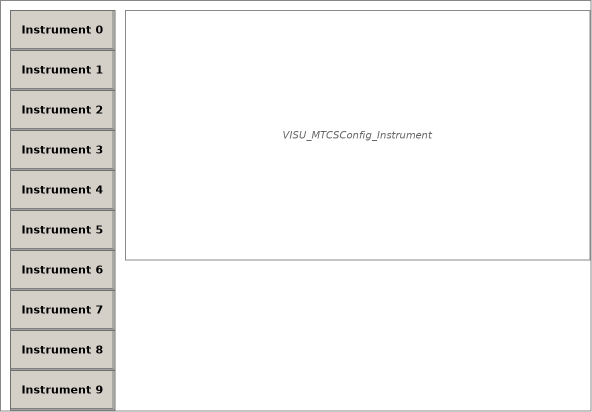
VISUALIZATION VISU_MTCSConfig_Instruments  // 592x412
VAR_IN_OUT
    active : MTCSInstrumentsConfig;
    editable : MTCSInstrumentsConfig;
	currentPosition : INT;
END_VAR
    Button (10,10 105x40), "Instrument 0", pressed state: currentPosition = 0
        OnMouseClick: execute { currentPosition := 0; }
    Button (10,50 105x40), "Instrument 1", pressed state: currentPosition = 1
        OnMouseClick: execute { currentPosition := 1; }
    Button (10,90 105x40), "Instrument 2", pressed state: currentPosition = 2
        OnMouseClick: execute { currentPosition := 2; }
    Button (10,130 105x40), "Instrument 3", pressed state: currentPosition = 3
        OnMouseClick: execute { currentPosition := 3; }
    Button (10,170 105x40), "Instrument 4", pressed state: currentPosition = 4
        OnMouseClick: execute { currentPosition := 4; }
    Button (10,210 105x40), "Instrument 5", pressed state: currentPosition = 5
        OnMouseClick: execute { currentPosition := 5; }
    Button (10,250 105x40), "Instrument 6", pressed state: currentPosition = 6
        OnMouseClick: execute { currentPosition := 6; }
    Button (10,290 105x40), "Instrument 7", pressed state: currentPosition = 7
        OnMouseClick: execute { currentPosition := 7; }
    Button (10,330 105x40), "Instrument 8", pressed state: currentPosition = 8
        OnMouseClick: execute { currentPosition := 8; }
    Button (10,370 105x40), "Instrument 9", pressed state: currentPosition = 9
        OnMouseClick: execute { currentPosition := 9; }
    Frame (125,10 465x250), frame switch variable: currentPosition
        shows VISU_MTCSConfig_Instrument(active := active.instrument0, editable := editable.instrument0)
        shows VISU_MTCSConfig_Instrument(active := active.instrument1, editable := editable.instrument1)
        shows VISU_MTCSConfig_Instrument(active := active.instrument2, editable := editable.instrument2)
        shows VISU_MTCSConfig_Instrument(active := active.instrument3, editable := editable.instrument3)
        shows VISU_MTCSConfig_Instrument(active := active.instrument4, editable := editable.instrument4)
        shows VISU_MTCSConfig_Instrument(active := active.instrument5, editable := editable.instrument5)
        shows VISU_MTCSConfig_Instrument(active := active.instrument6, editable := editable.instrument6)
        shows VISU_MTCSConfig_Instrument(active := active.instrument7, editable := editable.instrument7)
        shows VISU_MTCSConfig_Instrument(active := active.instrument8, editable := editable.instrument8)
        shows VISU_MTCSConfig_Instrument(active := active.instrument9, editable := editable.instrument9)
END_VISUALIZATION

(* stored: Version 1.1.0.1, ProductVersion 3.1.4019.2
   Visu VISU_MTCSConfig_Instruments: Id {d3acddf9-3f4c-4282-b9e9-74c943b482a6} *)
